% RSLogix 500 project P2 - Digital Filling Station.RSS, saved by version 8.30.00.16 %
PROJECT "PROJECT2"    % processor: Bul.1763 MicroLogix 1100 Series B %

PROGRAM FILES
  LAD 2 "MAIN"  3 rungs
  LAD 3 "IO"  8 rungs
  LAD 4 "CONTROLS"  7 rungs

DATA FILES
  O0 OUTPUT  4 elements
  I1 INPUT  6 elements
  S2 STATUS  66 elements
  B3 BINARY  2 elements
  T4 TIMER  3 elements
  C5 COUNTER  1 elements
  R6 CONTROL  1 elements
  N7 INTEGER  1 elements
  F8 FLOAT  1 elements

LADDER 2 "MAIN"
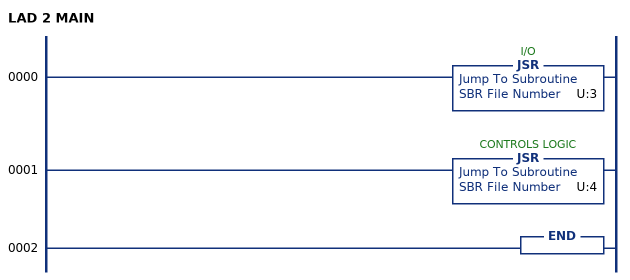
% Rung: 0 %
SOR JSR U:3 EOR
%   U:3  "I/O" %
% Rung: 1 %
SOR JSR U:4 EOR
%   U:4  "CONTROLS LOGIC" %
% Rung: 2 %
SOR END EOR

LADDER 3 "IO"
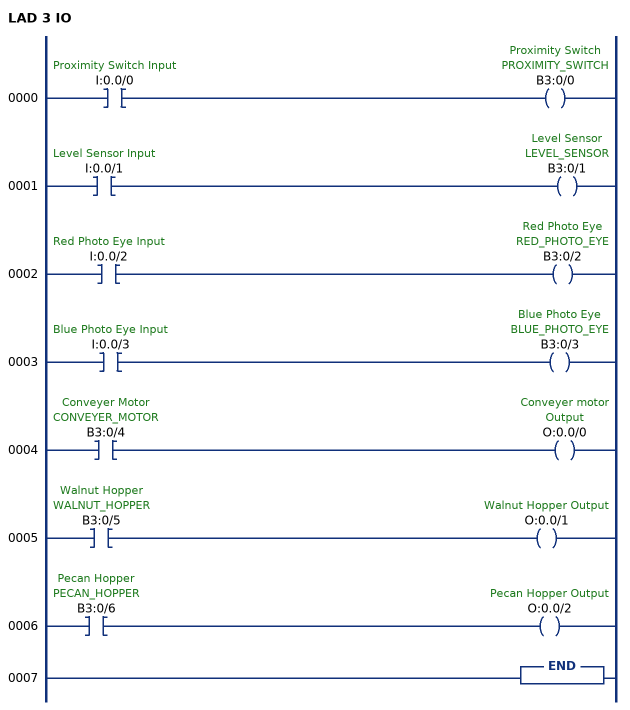
% Rung: 0 %
SOR XIC I:0.0/0 OTE B3:0/0 EOR
%   I:0.0/0  "Proximity Switch Input" %
%   B3:0/0  PROXIMITY_SWITCH  "Proximity Switch" %
% Rung: 1 %
SOR XIC I:0.0/1 OTE B3:0/1 EOR
%   I:0.0/1  "Level Sensor Input" %
%   B3:0/1  LEVEL_SENSOR  "Level Sensor" %
% Rung: 2 %
SOR XIC I:0.0/2 OTE B3:0/2 EOR
%   I:0.0/2  "Red Photo Eye Input" %
%   B3:0/2  RED_PHOTO_EYE  "Red Photo Eye" %
% Rung: 3 %
SOR XIC I:0.0/3 OTE B3:0/3 EOR
%   I:0.0/3  "Blue Photo Eye Input" %
%   B3:0/3  BLUE_PHOTO_EYE  "Blue Photo Eye" %
% Rung: 4 %
SOR XIC B3:0/4 OTE O:0.0/0 EOR
%   B3:0/4  CONVEYER_MOTOR  "Conveyer Motor" %
%   O:0.0/0  "Conveyer motor Output" %
% Rung: 5 %
SOR XIC B3:0/5 OTE O:0.0/1 EOR
%   B3:0/5  WALNUT_HOPPER  "Walnut Hopper" %
%   O:0.0/1  "Walnut Hopper Output" %
% Rung: 6 %
SOR XIC B3:0/6 OTE O:0.0/2 EOR
%   B3:0/6  PECAN_HOPPER  "Pecan Hopper" %
%   O:0.0/2  "Pecan Hopper Output" %
% Rung: 7 %
SOR END EOR

LADDER 4 "CONTROLS"
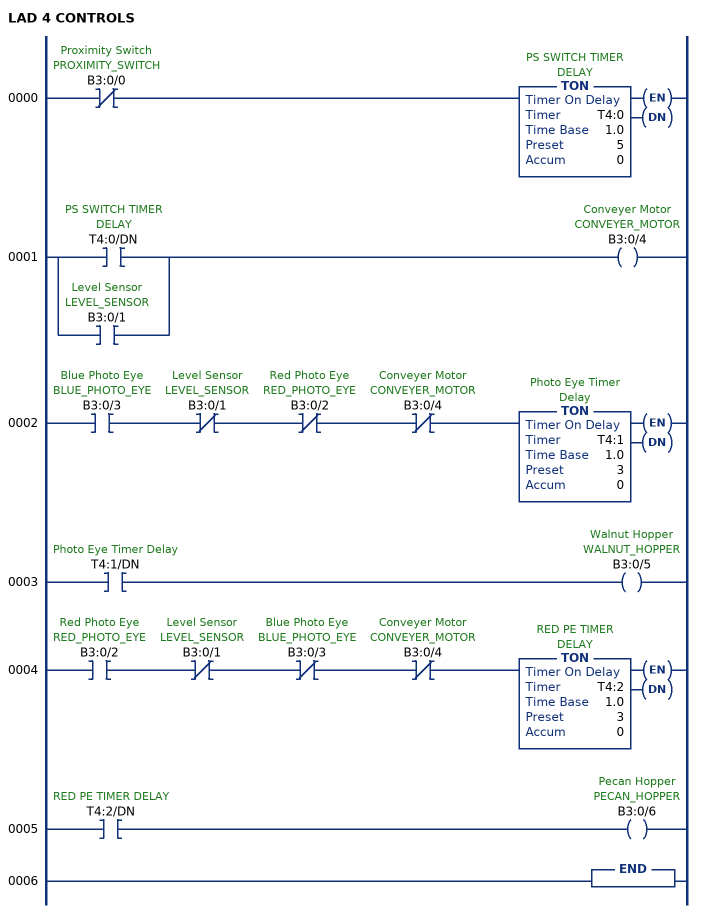
% Rung: 0 %
SOR XIO B3:0/0 TON T4:0 1.0 5 0 EOR
%   B3:0/0  PROXIMITY_SWITCH  "Proximity Switch" %
%   T4:0  "PS SWITCH TIMER DELAY" %
% Rung: 1 %
SOR BST XIC T4:0/DN NXB XIC B3:0/1 BND OTE B3:0/4 EOR
%   T4:0  "PS SWITCH TIMER DELAY" %
%   B3:0/1  LEVEL_SENSOR  "Level Sensor" %
%   B3:0/4  CONVEYER_MOTOR  "Conveyer Motor" %
% Rung: 2 %
SOR XIC B3:0/3 XIO B3:0/1 XIO B3:0/2 XIO B3:0/4 TON T4:1 1.0 3 0 EOR
%   B3:0/3  BLUE_PHOTO_EYE  "Blue Photo Eye" %
%   B3:0/1  LEVEL_SENSOR  "Level Sensor" %
%   B3:0/2  RED_PHOTO_EYE  "Red Photo Eye" %
%   B3:0/4  CONVEYER_MOTOR  "Conveyer Motor" %
%   T4:1  "Photo Eye Timer Delay" %
% Rung: 3 %
SOR XIC T4:1/DN OTE B3:0/5 EOR
%   T4:1  "Photo Eye Timer Delay" %
%   B3:0/5  WALNUT_HOPPER  "Walnut Hopper" %
% Rung: 4 %
SOR XIC B3:0/2 XIO B3:0/1 XIO B3:0/3 XIO B3:0/4 TON T4:2 1.0 3 0 EOR
%   B3:0/2  RED_PHOTO_EYE  "Red Photo Eye" %
%   B3:0/1  LEVEL_SENSOR  "Level Sensor" %
%   B3:0/3  BLUE_PHOTO_EYE  "Blue Photo Eye" %
%   B3:0/4  CONVEYER_MOTOR  "Conveyer Motor" %
%   T4:2  "RED PE TIMER DELAY" %
% Rung: 5 %
SOR XIC T4:2/DN OTE B3:0/6 EOR
%   T4:2  "RED PE TIMER DELAY" %
%   B3:0/6  PECAN_HOPPER  "Pecan Hopper" %
% Rung: 6 %
SOR END EOR

OTHER DOCUMENTED ADDRESSES
  B3:0/7  "Photo Eye Trigger"
  B3:0/8  "one shot 1"
  B3:0/9  "one shot 2"
  B3:1/0  "PS Trigger bit"
  T4:0/0  "PS SWITCH TIMER DELAY"
  T4:0/1  "Photo Eye Timer Delay"

DATA TABLE (non-zero values as saved)
DATA T4
% .PRE .ACC %
% T4:0 % 5 0
% T4:1 % 3 0
% T4:2 % 3 0
